INTERFACE I_MessageData

PROPERTY DirRoot : POINTER to string(255)
SET
END_SET
END_PROPERTY

PROPERTY ErrorIndex : reference to uint
SET
END_SET
END_PROPERTY

PROPERTY FileRoot : pointer to string(255)
SET
END_SET
END_PROPERTY

PROPERTY LocalTime : pointer to DT
SET
END_SET
END_PROPERTY

PROPERTY MessageIndex : reference to uint
SET
END_SET
END_PROPERTY

PROPERTY MsgList : pointer to ARRAY[1..GVL_MSG.MAX_MESSAGE] OF st_message
SET
END_SET
END_PROPERTY

END_INTERFACE

(* stored: Version 1.1.0.1
   Itf I_MessageData: Id {9cfc4b2d-eb33-49d8-836d-8e94c0b70b22}
   Property DirRoot: Id {af504870-47c6-4de1-a729-6e261778f0ab}
   Set Set: Id {73f02aae-f9fc-4fa1-b80a-bcf680962a9c}
   Property ErrorIndex: Id {0f078723-f3c4-4572-95ed-01d8d01566fc}
   Set Set: Id {b0ded0a9-2309-4548-bb79-c1793373ca53}
   Property FileRoot: Id {d7a46bd8-9281-49da-ac34-6a42c9f88e50}
   Set Set: Id {663785c6-41d9-4f5f-a4c0-f11e6c3b403e}
   Property LocalTime: Id {f0a26eed-7d5d-430b-9443-1396a99cb0ed}
   Set Set: Id {12a9862a-e6f4-42c9-8fe1-fb3f3ab06483}
   Property MessageIndex: Id {0d893ae0-6394-4921-859b-a3a8b9da532a}
   Set Set: Id {932df668-86b1-4feb-80d6-fe0962743268}
   Property MsgList: Id {2a9dafb5-5b29-47cf-8a16-2f5dd2de2c5b}
   Set Set: Id {7add3204-1f1e-4a7f-99f3-6c91e58cca7c} *)
